// TIA Portal V20 export
// export: Created 2026-09-14T11:29:00.3454864Z, ExportSetting None, DisplayName Totally Integrated Automation Portal, DisplayVersion V20, DisplayName TIA Portal Openness, DisplayVersion V20, DisplayName TIA Portal Version Control Interface, DisplayVersion V20, DisplayName STEP 7 Professional, DisplayVersion V20, DisplayName STEP 7 Safety, DisplayVersion V20, DisplayName WinCC Basic/Comfort/Advanced, DisplayVersion V20, DisplayName WinCC Unified, DisplayVersion V20
TYPE "LMQTT_typeTcpConnParamData"
   STRUCT
      useQdn : Bool;   // When TRUE, configure the connection for TCP over the fully qualified domain name
      hwIdentifier : HW_ANY;   // HW_ID of the PROFINET interface of the CPU
      connectionID : CONN_OUC;   // ID of the TCP connection
      qdnAdressBroker : String[254];   // URL of the MQTT Broker . Must end with a dot (".")
      ipAdressBroker : Array[0..3] of USInt;   // IP Address of the broker, e.g.: for the address "192.168.0.10"
      localPort : UInt := 0;   // Local port number of the CPU
      mqttPort : UInt := 1884;   // Remote port of the MQTT broker
      activateSecureConn : Bool;   // When TRUE, the communication is secured via TLS
      validateSubjectAlternateNameOfServer : Bool;   // Only for the client side. When TRUE, the IP address / QDN of the Broker is validated against the certificates SAN when the connection is established.
      idTlsServerCertificate : UDInt;   // Identifier of X.509 certificate (usually a CA certificate) to validate the authetication of the TLS server. Only relevant, if "activateSecureConn" is "true"
      idTlsOwnCertificate : UDInt;   // Identifier of own X.509 certificate to validate the own authetication against the TLS server. Only relevant, if "activateSecureConn" is "true" and the TLS server requests a client authentication
   END_STRUCT;
   // // ipAdressBroker[0] : "192"
   // // ipAdressBroker[1] : "168"
   // // ipAdressBroker[2] : "0"
   // // ipAdressBroker[3] : "10"
END_TYPE
